FUNCTION_BLOCK FbAlarm (* Блок предупреждений. *)
  (* Standard: 61499-1; Description: Блок предупреждений. Simple FB with one algorithm *)
  (* Version 2.2, 2026-03-20, VA, LIB_PLC *)
  (* Documentation:
  // Блок предупреждений. //          DbAlarm //    +-----------------+ //    |     FbAlarm     | // ->-|In        AlarmHi|->- //   -|LevelHi   AlarmLo|->- //   -|LevelLo          | //   -|TimeDelay        | //   -|Ts_ms            | //    +-----------------+
  *)
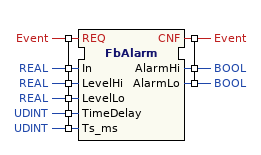
  EVENT_INPUT
    REQ WITH In, LevelHi, LevelLo, TimeDelay, Ts_ms; (* Normal Execution Request *)
  END_EVENT
  EVENT_OUTPUT
    CNF WITH AlarmHi, AlarmLo; (* Execution Confirmation *)
  END_EVENT
  VAR_INPUT
    In : REAL := 0.0; (* Входной сигнал. *)
    LevelHi : REAL := 0.0; (* Верхняя граница предупреждения. *)
    LevelLo : REAL := 0.0; (* Нижняя граница предупреждения. *)
    TimeDelay : UDINT := 0; (* Время задержки включения [мс]. *)
    Ts_ms : UDINT := 0; (* Шаг дискретизации по времени [мс]. *)
  END_VAR
  VAR_OUTPUT
    AlarmHi : BOOL := FALSE; (* Достигнут верхний предел. *)
    AlarmLo : BOOL := FALSE; (* Достигнут нижний предел. *)
  END_VAR
  VAR
    _AlarmHi : BOOL := FALSE; (* Достигнут верхний предел. *)
    _AlarmLo : BOOL := FALSE; (* Достигнут нижний предел. *)
    Timer1 : UDINT := 0; (* Текущее время таймер1 [мс]. *)
    Timer2 : UDINT := 0; (* Текущее время таймер1 [мс]. *)
  END_VAR
  EC_STATES
    REQ : REQ -> CNF;
  END_STATES
  ALGORITHM REQ IN ST:
// Верхний предел.
_AlarmHi := (In >= LevelHi);

// Таймер задержки включения для верхнего предела.
IF (TimeDelay > 0) THEN // Таймер включен.
	IF (_AlarmHi) THEN // На входе 1.
		IF (AlarmHi) THEN // На выходе 1.
			AlarmHi := TRUE;
		ELSE // На выходе 0.
			IF (Timer1 >= TimeDelay) THEN // Задержка включения закончилась.
				AlarmHi := TRUE;
			ELSE // Задержка включения активна.
				AlarmHi := FALSE;
				Timer1 := Timer1 + Ts_ms;
			END_IF;
		END_IF;
	ELSE // Если на входе 0 то на выходе тоже 0.
		AlarmHi := FALSE;
		Timer1 := 0;
	END_IF;
ELSE // Таймер выключен.
	AlarmHi := _AlarmHi;
	Timer1 := 0;
END_IF;

// Нижний предел.
_AlarmLo := (In <= LevelLo);

// Таймер задержки включения для нижнего предела.
IF (TimeDelay > 0) THEN // Таймер включен.
	IF (_AlarmLo) THEN // На входе 1.
		IF (AlarmLo) THEN // На выходе 1.
			AlarmLo := TRUE;
		ELSE // На выходе 0.
			IF (Timer2 >= TimeDelay) THEN // Задержка включения закончилась.
				AlarmLo := TRUE;
			ELSE // Задержка включения активна.
				AlarmLo := FALSE;
				Timer2 := Timer2 + Ts_ms;
			END_IF;
		END_IF;
	ELSE // Если на входе 0 то на выходе тоже 0.
		AlarmLo := FALSE;
		Timer2 := 0;
	END_IF;
ELSE // Таймер выключен.
	AlarmLo := _AlarmLo;
	Timer2 := 0;
END_IF;

// @COPYLEFT ALL WRONGS RESERVED :)
// Author: VA
// Contacts: DIY.PLC.314@gmail.com
// Date start LIB_PLC: 2014
// License: GNU GPL-2.0-or-later
// https://www.gnu.org/licenses/old-licenses/gpl-2.0.html
// https://www.youtube.com/watch?v=n1F_MfLRlX0
// https://www.youtube.com/@DIY_PLC
// https://github.com/DIYPLC/LIB_PLC
// https://oshwlab.com/diy.plc.314/PLC_HW1_SW1
// https://3dtoday.ru/3d-models/mechanical-parts/body/korpus-na-din-reiku
// https://t.me/DIY_PLC
  END_ALGORITHM
END_FUNCTION_BLOCK
